{attribute 'qualified_only'}
{attribute 'strict'}
TYPE E_FSM_AmeCltSq :
(
	IDLE,
	CREATE_MSG_TO_SEND,
	CALL_SEND_RCV_SQ,
	ERROR,
	DONE
);
END_TYPE

(* stored: Version 1.1.0.1
   DUT E_FSM_AmeCltSq: Id {a1905c1b-7beb-05e2-26b5-30c7047e48c0} *)
